// TIA Portal V16 export
// export: Created 2022-11-14T17:35:48.6639262Z, ExportSetting WithDefaults, DisplayName Totally Integrated Automation Portal, DisplayVersion V16, DisplayName TIA Portal Version Control Interface, DisplayVersion V16, DisplayName TIA Portal Openness, DisplayVersion V16, DisplayName STEP 7 Professional, DisplayVersion V16, DisplayName STEP 7 Safety, DisplayVersion V16, DisplayName WinCC Advanced, DisplayVersion V16
DATA_BLOCK "DB245_Program5"   // DB245
{ S7_Optimized_Access := 'FALSE' }
AUTHOR : Robopac
VERSION : 0.0
// stored: AutoNumber false, IsOnlyStoredInLoadMemory false, IsWriteProtectedInAS false
   VAR RETAIN
      Program5 { S7_SetPoint := 'True'} : "DatiProgramma";
   END_VAR
BEGIN
   Program5.Wrapping := TRUE;
   Program5.TopLenght := 500;
   Program5.TopRelease := 0;
   Program5.TopDown := 0;
   Program5.Top := 4;
   Program5.PressurePTime := 0;
   Program5.LifterTime := 0;
   Program5.RevOverContrast := 1;
   Program5.RopeEndCycle := 16#02;
   Program5.Spare4 := 16#01;
   Program5.RopeTime := 1500;
   Program5.RevOverClamp := 1;
   Program5.FilmForceFinalRev := 10;
   Program5.FilmPrestretchFinalRev := 100;
   Program5.ArmSpeed := 100;
   Program5.CarriageDown4Top := 500;
   Program5.TopDownTime := 1500;
   Program5.LapsUnderTop := 0;
   Program5.Spare6 := 0;
   Program5.Spare7 := 0;
   Program5.Spare8 := 0;
   Program5.Spare9 := 0;
   Program5.Spare10 := 0;
   Program5.Spare11 := 0;
   Program5.Spare12 := 0;
   Program5.Overlap0_1 := 0;
   Program5.Height1 := 130;
   Program5.Landmark1 := FALSE;
   Program5.Lifter1 := FALSE;
   Program5.SpareBit1H1 := FALSE;
   Program5.Airblower1 := TRUE;
   Program5.NextStep1 := TRUE;
   Program5.PressureP1 := TRUE;
   Program5.SpareByte2H1 := 16#00;
   Program5.Revolution1 := 1;
   Program5.RopeUnit1_1 := 16#01;
   Program5.RopeUnit1_2 := 16#01;
   Program5.FilmForce1 := 5;
   Program5.FilmPrestretch1 := 200;
   Program5.Spare3H1 := 0;
   Program5.Spare49 := 0;
   Program5.Spare50 := 0;
   Program5.Spare51 := 0;
   Program5.Spare52 := 0;
   Program5.Spare53 := 0;
   Program5.Overlap1_2 := 0;
   Program5.Height2 := 50;
   Program5.Landmark2 := FALSE;
   Program5.Lifter2 := FALSE;
   Program5.SpareBit1H2 := FALSE;
   Program5.Airblower2 := TRUE;
   Program5.NextStep2 := TRUE;
   Program5.PressureP2 := TRUE;
   Program5.SpareByte2H2 := 16#00;
   Program5.Revolution2 := 1;
   Program5.RopeUnit2_1 := 16#01;
   Program5.RopeUnit2_2 := 16#01;
   Program5.FilmForce2 := 20;
   Program5.FilmPrestretch2 := 200;
   Program5.Spare3H2 := 0;
   Program5.Spare54 := 0;
   Program5.Spare55 := 0;
   Program5.Spare56 := 0;
   Program5.Spare57 := 0;
   Program5.Spare58 := 0;
   Program5.Overlap2_3 := 100;
   Program5.Height3 := -50;
   Program5.Landmark3 := TRUE;
   Program5.Lifter3 := FALSE;
   Program5.SpareBit1H3 := FALSE;
   Program5.Airblower3 := TRUE;
   Program5.NextStep3 := TRUE;
   Program5.PressureP3 := TRUE;
   Program5.SpareByte2H3 := 16#00;
   Program5.Revolution3 := 2;
   Program5.RopeUnit3_1 := 16#01;
   Program5.RopeUnit3_2 := 16#01;
   Program5.FilmForce3 := 30;
   Program5.FilmPrestretch3 := 200;
   Program5.Spare3H3 := 0;
   Program5.Spare59 := 0;
   Program5.Spare60 := 0;
   Program5.Spare61 := 380;
   Program5.Spare62 := 2800;
   Program5.Spare63 := 0;
   Program5.Overlap3_4 := 100;
   Program5.Height4 := 100;
   Program5.Landmark4 := FALSE;
   Program5.Lifter4 := FALSE;
   Program5.SpareBit1H4 := FALSE;
   Program5.Airblower4 := TRUE;
   Program5.NextStep4 := TRUE;
   Program5.PressureP4 := TRUE;
   Program5.SpareByte2H4 := 16#00;
   Program5.Revolution4 := 3;
   Program5.RopeUnit4_1 := 16#02;
   Program5.RopeUnit4_2 := 16#02;
   Program5.FilmForce4 := 30;
   Program5.FilmPrestretch4 := 200;
   Program5.Spare3H4 := 0;
   Program5.Spare64 := 0;
   Program5.Spare65 := 0;
   Program5.Spare66 := 0;
   Program5.Spare67 := 0;
   Program5.Spare68 := 0;
   Program5.Overlap4_5 := 0;
   Program5.Height5 := 50;
   Program5.Landmark5 := FALSE;
   Program5.Lifter5 := FALSE;
   Program5.SpareBit1H5 := FALSE;
   Program5.Airblower5 := TRUE;
   Program5.NextStep5 := FALSE;
   Program5.PressureP5 := FALSE;
   Program5.SpareByte2H5 := 16#00;
   Program5.Revolution5 := 1;
   Program5.RopeUnit5_1 := 16#01;
   Program5.RopeUnit5_2 := 16#01;
   Program5.FilmForce5 := 30;
   Program5.FilmPrestretch5 := 200;
   Program5.Spare3H5 := 0;
   Program5.Spare69 := 0;
   Program5.Spare70 := 0;
   Program5.Spare71 := 0;
   Program5.Spare72 := 0;
   Program5.Spare73 := 0;
   Program5.Overlap5_6 := 100;
   Program5.Height6 := 50;
   Program5.Landmark6 := FALSE;
   Program5.Lifter6 := FALSE;
   Program5.SpareBit1H6 := FALSE;
   Program5.Airblower6 := TRUE;
   Program5.NextStep6 := FALSE;
   Program5.PressureP6 := FALSE;
   Program5.SpareByte2H6 := 16#00;
   Program5.Revolution6 := 2;
   Program5.RopeUnit6_1 := 16#02;
   Program5.RopeUnit6_2 := 16#01;
   Program5.FilmForce6 := 20;
   Program5.FilmPrestretch6 := 200;
   Program5.Spare3H6 := 0;
   Program5.Spare74 := 0;
   Program5.Spare75 := 0;
   Program5.Spare76 := 0;
   Program5.Spare77 := 0;
   Program5.Spare78 := 0;
   Program5.Overlap6_7 := 0;
   Program5.Height7 := 0;
   Program5.Landmark7 := FALSE;
   Program5.Lifter7 := FALSE;
   Program5.SpareBit1H7 := FALSE;
   Program5.Airblower7 := FALSE;
   Program5.NextStep7 := TRUE;
   Program5.PressureP7 := FALSE;
   Program5.SpareByte2H7 := 16#00;
   Program5.Revolution7 := 1;
   Program5.RopeUnit7_1 := 16#01;
   Program5.RopeUnit7_2 := 16#01;
   Program5.FilmForce7 := 0;
   Program5.FilmPrestretch7 := 100;
   Program5.Spare3H7 := 0;
   Program5.Spare79 := 0;
   Program5.Spare80 := 0;
   Program5.Spare81 := 0;
   Program5.Spare82 := 0;
   Program5.Spare83 := 0;
   Program5.Overlap7_8 := 0;
   Program5.Height8 := 0;
   Program5.Landmark8 := FALSE;
   Program5.Lifter8 := FALSE;
   Program5.SpareBit1H8 := FALSE;
   Program5.Airblower8 := FALSE;
   Program5.NextStep8 := TRUE;
   Program5.PressureP8 := FALSE;
   Program5.SpareByte2H8 := 16#00;
   Program5.Revolution8 := 1;
   Program5.RopeUnit8_1 := 16#01;
   Program5.RopeUnit8_2 := 16#01;
   Program5.FilmForce8 := 0;
   Program5.FilmPrestretch8 := 100;
   Program5.Spare3H8 := 0;
   Program5.Spare84 := 0;
   Program5.Spare85 := 0;
   Program5.Spare86 := 0;
   Program5.Spare87 := 0;
   Program5.Spare88 := 0;
   Program5.Overlap8_9 := 0;
   Program5.Height9 := 0;
   Program5.Landmark9 := FALSE;
   Program5.Lifter9 := FALSE;
   Program5.SpareBit1H9 := FALSE;
   Program5.Airblower9 := FALSE;
   Program5.NextStep9 := TRUE;
   Program5.PressureP9 := FALSE;
   Program5.SpareByte2H9 := 16#00;
   Program5.Revolution9 := 1;
   Program5.RopeUnit9_1 := 16#01;
   Program5.RopeUnit9_2 := 16#01;
   Program5.FilmForce9 := 0;
   Program5.FilmPrestretch9 := 100;
   Program5.Spare3H9 := 0;
   Program5.Spare89 := 0;
   Program5.Spare90 := 0;
   Program5.Spare91 := 0;
   Program5.Spare92 := 0;
   Program5.Spare93 := 0;
   Program5.Overlap9_10 := 0;
   Program5.Height10 := 0;
   Program5.Landmark10 := FALSE;
   Program5.Lifter10 := FALSE;
   Program5.SpareBit1H10 := FALSE;
   Program5.Airblower10 := FALSE;
   Program5.NextStep10 := FALSE;
   Program5.PressureP10 := FALSE;
   Program5.SpareByte2H10 := 16#00;
   Program5.Revolution10 := 1;
   Program5.RopeUnit10_1 := 16#01;
   Program5.RopeUnit10_2 := 16#01;
   Program5.FilmForce10 := 0;
   Program5.FilmPrestretch10 := 100;
   Program5.Spare3H10 := 0;
   Program5.Spare94 := 0;
   Program5.Spare95 := 0;
   Program5.Spare96 := 0;
   Program5.Spare97 := 0;
   Program5.Spare98 := 0;
   Program5.Overlap10_11 := 0;
   Program5.Height11 := 0;
   Program5.Landmark11 := FALSE;
   Program5.Lifter11 := FALSE;
   Program5.SpareBit1H11 := FALSE;
   Program5.Airblower11 := FALSE;
   Program5.NextStep11 := TRUE;
   Program5.PressureP11 := FALSE;
   Program5.SpareByte2H11 := 16#00;
   Program5.Revolution11 := 1;
   Program5.RopeUnit11_1 := 16#01;
   Program5.RopeUnit11_2 := 16#01;
   Program5.FilmForce11 := 0;
   Program5.FilmPrestretch11 := 100;
   Program5.Spare3H11 := 0;
   Program5.Spare99 := 0;
   Program5.Spare100 := 0;
   Program5.Spare101 := 0;
   Program5.Spare102 := 0;
   Program5.Spare103 := 0;
   Program5.Overlap11_12 := 0;
   Program5.Height12 := 0;
   Program5.Landmark12 := FALSE;
   Program5.Lifter12 := FALSE;
   Program5.SpareBit1H12 := FALSE;
   Program5.Airblower12 := FALSE;
   Program5.NextStep12 := FALSE;
   Program5.PressureP12 := FALSE;
   Program5.SpareByte2H12 := 16#00;
   Program5.Revolution12 := 1;
   Program5.RopeUnit12_1 := 16#01;
   Program5.RopeUnit12_2 := 16#01;
   Program5.FilmForce12 := 0;
   Program5.FilmPrestretch12 := 100;
   Program5.Spare3H12 := 0;
   Program5.Spare104 := 0;
   Program5.Spare105 := 0;
   Program5.Spare106 := 0;
   Program5.Spare107 := 0;
   Program5.Spare108 := 0;
END_DATA_BLOCK
